PROGRAM MAIN
VAR	

	// ========= System Control / FSM Variables =========
	
	MainCommands 		: MainCommands_typ; 		// command struct for cycling thru the state machine
	MainState    		: MainStateMachine_enum;   	// enumeration for the Main state machine
	System				: Mediator;					// System-level control object
	RecoveryComplete	: BOOL;						// flag tracking the completeness of start-up recovery

	// ========= Linked NC Variables & References =========
	
	Mover    			: ARRAY[1..GVL.NUM_MOVERS] OF Mover; 	// instantiation of Mover objects. Matches the number of movers on the system
	
	// ========= Objectives & Parameters =========

	ParameterSet		: MotionParameters_typ;
	
	MoverList			: ARRAY[0..GVL.NUM_MOVERLISTS-1] OF MoverList;
	PositionTrigger		: ARRAY[0..GVL.NUM_POSITIONTRIGGERS-1] OF PositionTrigger;
	Station				: ARRAY[0..GVL.NUM_STATIONS-1] OF Station;
	Track				: ARRAY[0..GVL.NUM_TRACKS] OF Track;
	Zone				: ARRAY[0..GVL.NUM_ZONES-1] OF Zone;
	
    // ========= Helper, State, & Index Variables =========
	
    i                	: UINT; 	// index variable; gets reused in various FOR loops
    n                	: UINT; 	// secondary index variable, for enabling movers
	
	// ========= Example Application Variables =========

    nextStation 			: USINT := 4;
                    	
    lowVelocity    			: LREAL := 200;  	// mm/s
    mediumVelocity 			: LREAL := 800;  	// mm/s
    highVelocity   			: LREAL := 1200; 	// mm/s
	
	StationTimer 			: ARRAY[0..GVL.NUM_STATIONS] OF TON; // timer blocks, for station dwells
	InitialParameterSet		: MotionParameters_typ;
	
END_VAR


CASE MainState OF
	MainStateMachine_enum.MS_DISABLED: // ------------------------------------------
	
		// XTS is idle. Motive power is disabled.	
		IF MainCommands.Enable THEN
			MainCommands.Disable			:= FALSE;
			MainCommands.Stop				:= FALSE;
			MainState						:= MainStateMachine_enum.MS_INITIALIZING;
		END_IF

	MainStateMachine_enum.MS_INITIALIZING: // --------------------------------------
	
		Registering();			// Add all objectives & movers to the system-level Mediator object
		Initializing();			// Set basic application parameters for the objects
			
		System.CompleteMoverList.EnableAll();
		System.CompleteMoverList.ActivateAllTrack( Track[1] );
		
		IF System.CompleteMoverList.IsAllTrackReady AND System.CompleteMoverList.IsAllMoversReady THEN
			MainState	:= MainStateMachine_enum.MS_ENABLED;
		END_IF
		
		IF MainCommands.Disable THEN
			MainCommands.Enable	:= FALSE;
			System.CompleteMoverList.DisableAll();
			MainState			:= MainStateMachine_enum.MS_DISABLING;
		END_IF
	
	MainStateMachine_enum.MS_ENABLED:	// -------------------------------------------
	
		// Check for system ready or disable command
		IF MainCommands.Start AND system.AllMotorModulesReady AND system.GroupEnabled THEN
			MainState			:= MainStateMachine_enum.MS_ONESHOT_RECOVER;
		ELSIF MainCommands.Disable THEN
			MainCommands.Enable	:= FALSE;
			System.CompleteMoverList.HaltAll();
			MainState			:= MainStateMachine_enum.MS_STOPPING;
			
		END_IF
		
	MainStateMachine_enum.MS_ONESHOT_RECOVER: // -----------------------------------------------
		// call the one-shot recovery state
		RecoverOneshot();
		
		// immediately continue to recover state
		MainState := MainStateMachine_enum.MS_RECOVERING;
		
	MainStateMachine_enum.MS_RECOVERING: // -----------------------------------------------
		// reset the recovering complete flag
		RecoveryComplete := FALSE;
		// call the recovering logic (sets complete flag when ready
		Recovering();
		
		// test for errors, commands or recovery complete
		IF System.GroupError THEN
			// stop on group error user must go through disable/enable to recover
			MainCommands.Start	:= FALSE;
			MainState 			:= MainStateMachine_enum.MS_STOPPING;
		ELSIF MainCommands.Stop THEN
            MainCommands.Start 	:= FALSE;
			System.CompleteMoverList.HaltAll();
            MainState         	:= MainStateMachine_enum.MS_STOPPING;
        ELSIF MainCommands.Disable THEN
            MainCommands.Enable := FALSE;
			System.CompleteMoverList.HaltAll();
            MainState           := MainStateMachine_enum.MS_STOPPING;
		ELSIF RecoveryComplete THEN
			// recovery sequence is complete, move on to run state
			MainState			:= MainStateMachine_enum.MS_RUN;
        END_IF
	
	MainStateMachine_enum.MS_RUN: // -----------------------------------------------
		// call the station logic
		StationLogic();
		
		// check for errors or other commands
        IF System.GroupError THEN
			// stop on group error user must go through disable/enable to recover
			MainCommands.Start	:= FALSE;
			MainState 			:= MainStateMachine_enum.MS_STOPPING;
		ELSIF MainCommands.Stop THEN
            MainCommands.Start 	:= FALSE;
			System.CompleteMoverList.HaltAll();
            MainState         	:= MainStateMachine_enum.MS_STOPPING;
        ELSIF MainCommands.Disable THEN
            MainCommands.Enable := FALSE;
			System.CompleteMoverList.HaltAll();
            MainState           := MainStateMachine_enum.MS_STOPPING;
        END_IF
		
	MainStateMachine_enum.MS_STOPPING:
	
		IF System.CompleteMoverList.IsAllMoversHalted THEN
			MainState			:= MainStateMachine_enum.MS_STOPPED;
		END_IF
		
	MainStateMachine_enum.MS_STOPPED: // -------------------------------------------
	
	    IF MainCommands.Disable THEN
            MainCommands.Enable 	:= FALSE;
			MainCommands.Start		:= FALSE;
			MainCommands.Stop		:= FALSE;
			System.CompleteMoverList.DisableAll();
            MainState           	:= MainStateMachine_enum.MS_DISABLING;
        ELSIF MainCommands.Start THEN
            MainCommands.Stop 		:= FALSE;
            MainState         		:= MainStateMachine_enum.MS_ENABLED;
        END_IF
		
	MainStateMachine_enum.MS_DISABLING: // -------------------------------------------
	
		IF System.CompleteMoverList.IsAllMoversDisabled THEN
			MainState			:= MainStateMachine_enum.MS_DISABLED;
		END_IF
		
	MainStateMachine_enum.MS_ERROR: // ---------------------------------------------
	MainStateMachine_enum.MS_DEBUG: // ---------------------------------------------	
	

END_CASE

System.Cyclic();

ACTION Initializing:


	// Initialize station positions
	Station[0].Position 		:= 5;
	Station[1].Position 		:= 750;
	Station[2].Position 		:= 1200;
	Station[3].Position 		:= 1300;
	Station[4].Position 		:= 1400;

	PositionTrigger[0].Position := 1500;
	PositionTrigger[1].Position := 2000;
	PositionTrigger[2].Position := 3500;

	Zone[0].StartPosition		:= 3750;
	Zone[0].EndPosition   		:= 750;

	Zone[1].StartPosition 		:= 750;
	Zone[1].EndPosition   		:= 1750;

	Zone[2].StartPosition 		:= 1750;
	Zone[2].EndPosition   		:= 2750;

	Zone[3].StartPosition		:= 2750;
	Zone[3].EndPosition   		:= 3750;

	InitialParameterSet.Velocity		:= 1000;		// mm/s
	InitialParameterSet.Acceleration	:= 10_000;		// mm/s2
	InitialParameterSet.Deceleration	:= 10_000;		// mm/s2
	InitialParameterSet.Jerk			:= 100_000;		// mm/s3
	InitialParameterSet.Gap				:= 85;			// mm
	InitialParameterSet.Direction		:= mcDirectionPositive;	
	
	System.CompleteMoverList.ApplyAllParameterSet( InitialParameterSet );
END_ACTION

ACTION Recovering:
// this state is called until all movers have completed their desired recovery tasks

// wait for all movers to reach the standstill state and one mover at station 0
IF (System.CompleteMoverList.IsAllMoversHalted and Station[0].MoverInPosition) THEN
	RecoveryComplete := TRUE;
END_IF
END_ACTION

ACTION RecoverOneshot:
// this action is called one time after the start command is issued
// it is intended to provide a single command to each mover to facilitate recovery
// other commands such as resetting counters and timers should also be carried out here

// send all movers to station 0
System.CompleteMoverList.SetAllVelocity(mediumVelocity).MoveAllToStation( Station[0] );
System.ResetStatistics();

// Reinit nextStation
nextStation := 4;
END_ACTION

ACTION Registering:
	

		// Add all Movers to the Mediator
		FOR i := 1 TO GVL.NUM_MOVERS DO
			System.AddMover( Mover[i] );
		END_FOR
	
		// Add all Mover Lists to the Mediator
		FOR i := 0 TO GVL.NUM_MOVERLISTS - 1 DO
			System.AddMoverList( MoverList[i] );
		END_FOR
		
		// Add all PositionTriggers to the Mediator
		FOR i := 0 TO GVL.NUM_POSITIONTRIGGERS - 1 DO
			System.AddPositionTrigger( PositionTrigger[i] );
			PositionTrigger[i].SetTrack(Track[1]);
		END_FOR
		
		// Add all Stations to the Mediator
		FOR i := 0 TO GVL.NUM_STATIONS - 1 DO
			System.AddStation( Station[i] );
			Station[i].SetTrack(Track[1]);
		END_FOR
		
		// Add all Tracks to the Mediator
		// note track zero is a special case, so the loop is one larger than the rest of the initalization loops
		FOR i := 0 TO GVL.NUM_TRACKS DO
			Track[i].Id := UINT_TO_INT(i);
			System.AddTrack( Track[i] );
		END_FOR
		
		// Add all Zones to the Mediator
		FOR i := 0 TO GVL.NUM_ZONES - 1 DO
			System.AddZone( Zone[i] );
			Zone[i].SetTrack(Track[1]);
		END_FOR
END_ACTION

ACTION StationLogic:
		(*Mover routing logic should be written here to define the system's operating behavior.
		Station implementations, Position Trigger logic, etc. In general, you can remove the example code
		here down to the short line break that looks like this: // ============= *)
	
        // Station 0 Logic
        IF Station[0].MoverInPosition THEN
            StationTimer[0](IN := TRUE, PT := T#1000MS);
            IF StationTimer[0].Q THEN
                Station[0].CurrentMover.SetVelocity(mediumVelocity);
                Station[0].CurrentMover.MoveToStation(Station[1]);
            END_IF
        ELSE
            StationTimer[0](IN := FALSE);
        END_IF
		
        // Station 1 Logic		
        IF Station[1].MoverInPosition THEN
            StationTimer[1](IN := TRUE, PT := T#250MS);
            IF StationTimer[1].Q THEN
                Station[1].CurrentMover.SetVelocity(mediumVelocity);
                Station[1].CurrentMover.MoveToStation(Station[nextStation]);
                nextStation := nextStation - 1;
                IF nextStation = 1 THEN
                    nextStation := 4;
                END_IF
            END_IF
        ELSE
            StationTimer[1](IN := FALSE);
        END_IF
		
		// Group of Stations 2, 3, and 4 Logic
        IF Station[2].MoverInPosition AND Station[3].MoverInPosition AND Station[4].MoverInPosition THEN
            StationTimer[2](IN := TRUE, PT := T#750MS);
            IF StationTimer[2].Q THEN
				StationTimer[2](IN := FALSE);

                Station[2].CurrentMover.MoveVelocity(500);
                Station[3].CurrentMover.MoveVelocity(500);
                Station[4].CurrentMover.MoveVelocity(500);
            END_IF
        END_IF
		
        // Position Trigger 0 Logic
        IF PositionTrigger[0].MoverPassedPosition THEN
            PositionTrigger[0].CurrentMover.SetVelocity(lowVelocity);
            PositionTrigger[0].MuteCurrent();
        END_IF
		
        // Position Trigger 1 Logic
        IF PositionTrigger[1].MoverPassedPosition THEN
			PositionTrigger[1].CurrentMover.SetAcceleration(5E2);
            PositionTrigger[1].CurrentMover.SetVelocity(highVelocity);
            PositionTrigger[1].MuteCurrent();
        END_IF

		// Position Trigger 2 Logic
        IF PositionTrigger[2].MoverPassedPosition THEN
			PositionTrigger[2].CurrentMover.SetAcceleration(1E4);
            PositionTrigger[2].CurrentMover.SetVelocity(lowVelocity);
            PositionTrigger[2].CurrentMover.MoveToStation(Station[0]);
            PositionTrigger[2].MuteCurrent();
        END_IF
END_ACTION

END_PROGRAM

(* stored: Version 1.1.0.1, ProductVersion 3.1.4026.8
   POU MAIN: Id {c992ed33-41fe-02c4-17ef-23123b9a5b23}, SpecialFunc None
   Action Initializing: Id {77eee1d6-568e-0448-2c64-a85af70fbf71}
   Action Recovering: Id {43063827-0598-00b7-2079-e6fbfd8a6aff}
   Action RecoverOneshot: Id {7eb1f3e7-2df1-00d5-25c0-031445570e00}
   Action Registering: Id {ef3ef836-2b88-0099-2899-1cd10004220b}
   Action StationLogic: Id {ad15b1d3-f9a4-013e-29dd-5430b02980cb} *)
